// TIA Portal V15.1 export
// export: Created 2020-06-12T07:35:41.6474609Z, ExportSetting None, DisplayName Totally Integrated Automation Portal, DisplayVersion V15.1, DisplayName TIA Portal Openness, DisplayVersion V15.1, DisplayName STEP 7 Professional, DisplayVersion V15.1, DisplayName STEP 7 Safety, DisplayVersion V15.1, DisplayName WinCC Advanced, DisplayVersion V15.1
FUNCTION "Common" : Void   // FC30, FBD
{ S7_Optimized_Access := 'TRUE' }
AUTHOR : atec
FAMILY : COMMON
NAME : Common
VERSION : 1.0
// stored: AutoNumber false, SetENOAutomatically False
   VAR_TEMP
      tWarnStartReq : Bool;
   END_VAR
   VAR_TEMP   // added for the SCL form of the ladder/FBD networks
      _w1 : Bool;
      _w2 : Bool;
      _w3 : Bool;
   END_VAR
BEGIN

REGION Network 1: System general: Power OK / Spannungsversorgung OK
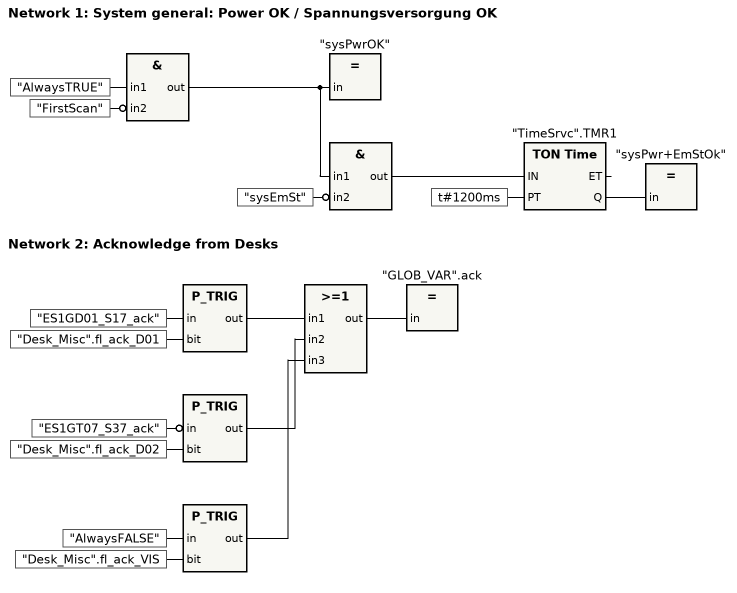
   "sysPwrOK" := "AlwaysTRUE" AND NOT "FirstScan";
   "TimeSrvc".TMR1.TON(IN := "sysPwrOK" AND NOT "sysEmSt", PT := t#1200ms);
   "sysPwr+EmStOk" := "TimeSrvc".TMR1.Q;
END_REGION

REGION Network 2: Acknowledge from Desks
   // TO REPLACE "MELT_CMD".ES1SZ1_horn_ack
   #_w1 := "ES1GD01_S17_ack" AND NOT "Desk_Misc".fl_ack_D01;   // rising edge
   "Desk_Misc".fl_ack_D01 := "ES1GD01_S17_ack";
   #_w2 := NOT "ES1GT07_S37_ack" AND NOT "Desk_Misc".fl_ack_D02;   // rising edge
   "Desk_Misc".fl_ack_D02 := NOT "ES1GT07_S37_ack";
   #_w3 := "AlwaysFALSE" AND NOT "Desk_Misc".fl_ack_VIS;   // rising edge
   "Desk_Misc".fl_ack_VIS := "AlwaysFALSE";
   "GLOB_VAR".ack := #_w1 OR #_w2 OR #_w3;
END_REGION
END_FUNCTION
